FUNCTION_BLOCK INTERNAL FB_SimMovitracFSM
VAR_INPUT
	bControllerInhibit	: BOOL;
	bRapidStop			: BOOL;
	bStop				: BOOL;
	bHoldControl		: BOOL;
END_VAR
VAR_OUTPUT
	eState			: E_SimMovitracState := E_SimMovitracState.ControllerInhibit;	
END_VAR

(* Statemachine *)	
	CASE eState OF	
		E_SimMovitracState.ControllerInhibit: ControllerInhibit();		
		E_SimMovitracState.RapidStop:	RapidStop();
		E_SimMovitracState.Halt: Halt();
		E_SimMovitracState.HoldControl: HoldControl();
		E_SimMovitracState.Enable: Enable();
	END_CASE

METHOD INTERNAL ControllerInhibit
VAR_INPUT
END_VAR
(*to RapidStop*)	
	IF NOT bControllerInhibit THEN
		eState := E_SimMovitracState.RapidStop;
	END_IF
END_METHOD

METHOD INTERNAL Enable
VAR_INPUT
END_VAR
(*to ControllerInhibit*)	
	IF bControllerInhibit THEN
		eState := E_SimMovitracState.ControllerInhibit;
		RETURN;
	END_IF

(*to RapidStop*)	
	IF NOT bRapidStop THEN
		eState := E_SimMovitracState.RapidStop;
		RETURN;
	END_IF
	
(*to Halt*)	
	IF NOT bStop THEN
		eState := E_SimMovitracState.Halt;
		RETURN;
	END_IF
	
(*to HoldControl*)	
	IF bHoldControl THEN
		eState := E_SimMovitracState.HoldControl;
	END_IF
END_METHOD

METHOD INTERNAL Halt
VAR_INPUT
END_VAR
(*to ControllerInhibit*)	
	IF bControllerInhibit THEN
		eState := E_SimMovitracState.ControllerInhibit;
		RETURN;
	END_IF

(*to RapidStop*)	
	IF NOT bRapidStop THEN
		eState := E_SimMovitracState.RapidStop;
		RETURN;
	END_IF
	
(*to HoldControl*)	
	IF bStop AND bHoldControl THEN
		eState := E_SimMovitracState.HoldControl;
		RETURN;
	END_IF

(*to Enable*)	
	IF bStop AND NOT bHoldControl THEN
		eState := E_SimMovitracState.Enable;
	END_IF
END_METHOD

METHOD INTERNAL HoldControl
VAR_INPUT
END_VAR
(*to ControllerInhibit*)	
	IF bControllerInhibit THEN
		eState := E_SimMovitracState.ControllerInhibit;
		RETURN;
	END_IF

(*to RapidStop*)	
	IF NOT bRapidStop THEN
		eState := E_SimMovitracState.RapidStop;
		RETURN;
	END_IF
	
(*to Halt*)	
	IF NOT bStop THEN
		eState := E_SimMovitracState.Halt;
		RETURN;
	END_IF
	
(*to Enable*)	
	IF NOT bHoldControl THEN
		eState := E_SimMovitracState.Enable;
	END_IF
END_METHOD

PROPERTY nState : E_SimMovitracState
GET
nState := eState;
END_GET
SET
eState := nState;
END_SET
END_PROPERTY

METHOD INTERNAL RapidStop
VAR_INPUT
END_VAR
(*to ControllerInhibit*)	
	IF bControllerInhibit THEN
		eState := E_SimMovitracState.ControllerInhibit;
		RETURN;
	END_IF

(*to Halt*)	
	IF bRapidStop THEN
		eState := E_SimMovitracState.Halt;
	END_IF
END_METHOD

END_FUNCTION_BLOCK

(* stored: Version 1.1.0.1, ProductVersion 3.1.4024.12
   POU FB_SimMovitracFSM: Id {13dfd547-1e98-0721-03fa-b95e41d349dd}, SpecialFunc None
   Method ControllerInhibit: Id {5b23a47f-a970-0c02-213c-2d154d590752}
   Method Enable: Id {178a8ed2-e4ec-02f0-272d-23f6afe6b876}
   Method Halt: Id {1439a7d3-7070-0541-1e83-a29773d45bf0}
   Method HoldControl: Id {cb7c0b11-0bc1-066b-0a35-3dbaf383a4dd}
   Property nState: Id {5b9e7a90-e13f-0d86-1112-6f77d141474c}
   Get Get: Id {8f8745ba-3fa1-05b0-01e5-29dfb0174d79}
   Set Set: Id {2c4f2a99-ebac-031c-178d-eca0dd67c5b6}
   Method RapidStop: Id {1fbc26e3-1fa4-061a-051e-8d9943ff0fdb} *)
